TEXTLIST KLoadMode
  0 = 'Suction'
  1 = 'Position'
  2 = 'Position+Torque'
   = ''
END_TEXTLIST

(* stored: Version 1.1.0.1, ProductVersion 3.1.4024.11
   TextList KLoadMode: Id {2ac652a8-947a-47f2-a69f-40b94ada0a77} *)
